// TIA Portal V19 export
TYPE "PathTestSignal"
// stored: Access Published
   STRUCT
      TestRequired : Bool;   // Path test required
      TestRunning : Bool;   // Path test running
      TestRunCmd : Bool;   // Path test run command
   END_STRUCT;
END_TYPE
